FUNCTION_BLOCK FB_DeformationPointFIFO
VAR_OUTPUT
	nCount    : UINT;                 // Fill level
END_VAR
VAR
	sBuffer 	: ARRAY[0..(MAX_BUFFER_SIZE-1)] OF ST_DeformationPoint;
	nHeadPtr  : UINT := 0;            // Point to the first non-empty idx
	nTailPtr  : UINT := 0;            // Pointer to the first free idx
  _bError    : BOOL;
END_VAR
VAR CONSTANT
	MAX_BUFFER_SIZE   : UINT := 1000;  // max. buffer size
	BUFFER_ITEM_SIZE  : UINT := SIZEOF(ST_DeformationPoint)/4; // Divide by 4 as we packed the ST_POINT with 32bits steps
END_VAR


(* now done async in method, this was dangerous...
// FIFO level
IF nTailPtr <= nHeadPtr THEN
	nCount := nHeadPtr - nTailPtr;
ELSE
	nCount := MAX_BUFFER_SIZE + nHeadPtr - nTailPtr;
END_IF
*)

PROPERTY bError : BOOL
GET
bError := _bError;
END_GET
END_PROPERTY

(*
  Get point from fifo queue. 
  :return: TRUE on success
*)
METHOD Pop : BOOL
VAR_OUTPUT
	sGridPoint : ST_DeformationPoint;
END_VAR
IF nCount = 0 THEN
  F_LogError('FB_DeformationPointFIFO is empty, cannot return an element');
  _bError := TRUE; 
  RETURN;
END_IF

sGridPoint := sBuffer[nTailPtr];
nTailPtr := (nTailPtr + 1) MOD MAX_BUFFER_SIZE;
nCount := nCount - 1;
_bError := FALSE;
Pop := TRUE;
END_METHOD

(*
  Add a new point to the fifo queue.
  :return: TRUE on success.
*)
METHOD Push : BOOL
VAR_INPUT
	sNewPoint : ST_DeformationPoint;
END_VAR
IF nCount >= MAX_BUFFER_SIZE THEN
  F_LogError('FB_DeformationPointFIFO overflow, element ignored');
  _bError := TRUE;
  RETURN;
END_IF

sBuffer[nHeadPtr] := sNewPoint;
nHeadPtr := (nHeadPtr + 1) MOD MAX_BUFFER_SIZE;
nCount := nCount + 1;
_bError := FALSE;
Push := TRUE;
END_METHOD

METHOD Reset : BOOL
VAR_INPUT
END_VAR
nTailPtr := 0;
nHeadPtr := 0;
nCount := 0;
_bError := 0;
END_METHOD

END_FUNCTION_BLOCK

(* stored: Version 1.1.0.1, ProductVersion 3.1.4024.3
   POU FB_DeformationPointFIFO: Id {1c595d80-10e4-4767-bff8-0ee27da948ff}, SpecialFunc None
   Property bError: Id {2c0c8ac4-7879-4f9b-ac5a-6b595df476ae}
   Get Get: Id {d3e01224-9b76-4141-90f9-3c5b23c5a32b}
   Method Pop: Id {1407fd01-3e55-406d-afdb-7f3babec0896}
   Method Push: Id {ad235f3c-7a4c-4435-a3a6-ef3cf622a917}
   Method Reset: Id {49c6e9ec-a40e-42ed-96a8-eff7c0fd072c} *)
